// Mitsubishi GX Works2 project: 西松湘南道路1号機   PLC: Q03UDV
// 鹿島外環ロスゼロ

PROGRAM SIMLAT
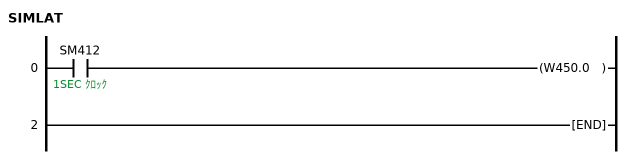
0     LD      SM412  ; 1SEC ｸﾛｯｸ
      OUT     W450.0
2     END
END_PROGRAM

PROGRAM FLEXPIWI
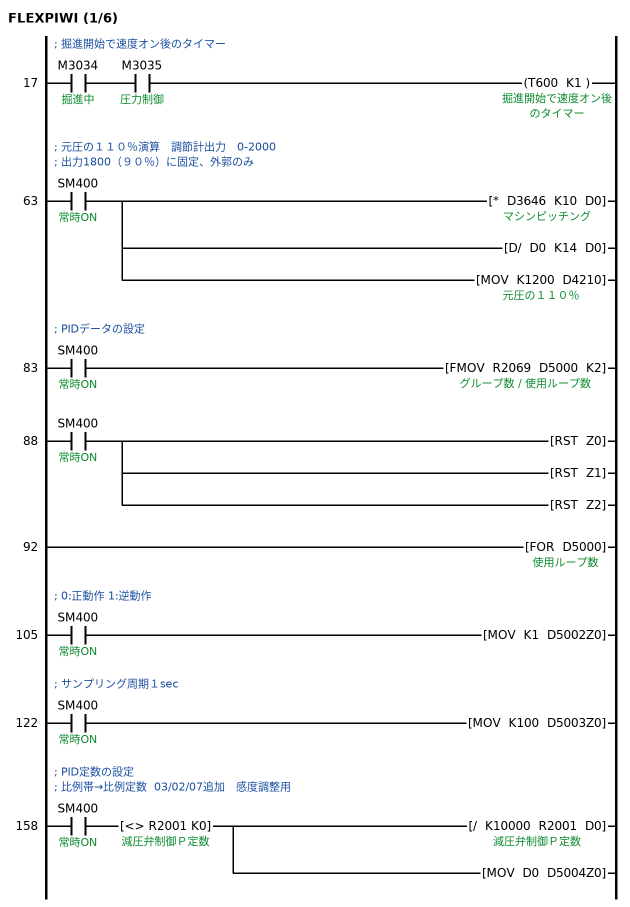
; 掘進開始で速度オン後のタイマー
17    LD      M3034  ; 掘進中
      AND     M3035  ; 圧力制御
      OUT     T600 K1  ; 掘進開始で速度オン後のタイマー
; 元圧の１１０％演算　調節計出力　0-2000
; 出力1800（９０％）に固定、外郭のみ
63    LD      SM400  ; 常時ON
      *       D3646 K10 D0  ; マシンピッチング
      D/      D0 K14 D0
      MOV     K1200 D4210  ; 元圧の１１０％
; PIDデータの設定
83    LD      SM400  ; 常時ON
      FMOV    R2069 D5000 K2  ; グループ数 / 使用ループ数
88    LD      SM400  ; 常時ON
      RST     Z0
      RST     Z1
      RST     Z2
92    FOR     D5000
; 0:正動作 1:逆動作
105   LD      SM400  ; 常時ON
      MOV     K1 D5002Z0
; サンプリング周期１sec
122   LD      SM400  ; 常時ON
      MOV     K100 D5003Z0
; PID定数の設定
; 比例帯→比例定数  03/02/07追加　感度調整用
158   LD      SM400  ; 常時ON
      AND<>   R2001 K0  ; 減圧弁制御Ｐ定数
      /       K10000 R2001 D0
      MOV     D0 D5004Z0
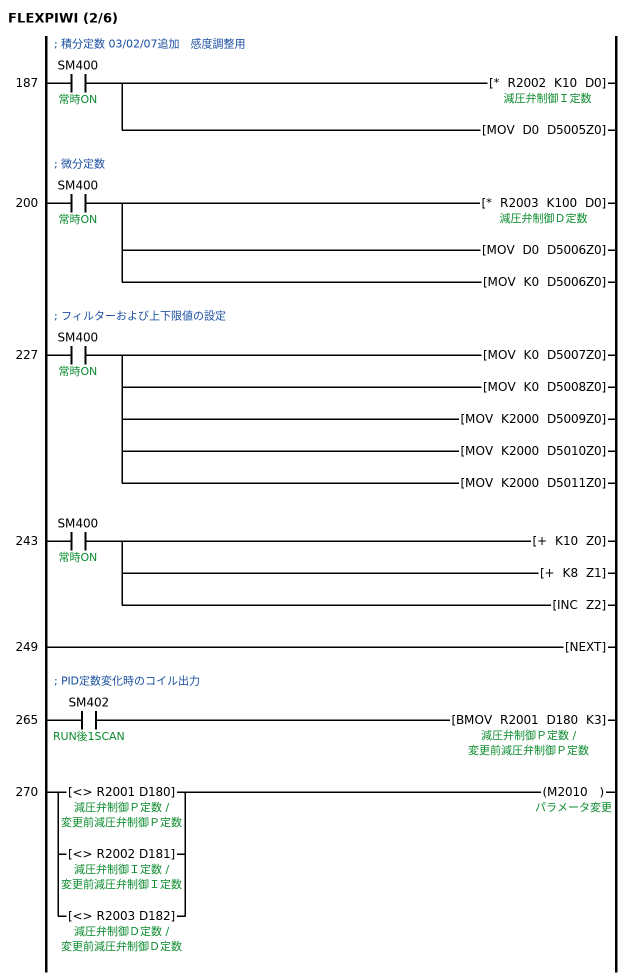
; 積分定数 03/02/07追加　感度調整用
187   LD      SM400  ; 常時ON
      *       R2002 K10 D0  ; 減圧弁制御Ｉ定数
      MOV     D0 D5005Z0
; 微分定数
200   LD      SM400  ; 常時ON
      *       R2003 K100 D0  ; 減圧弁制御Ｄ定数
      MOV     D0 D5006Z0
      MOV     K0 D5006Z0
; フィルターおよび上下限値の設定
227   LD      SM400  ; 常時ON
      MOV     K0 D5007Z0
      MOV     K0 D5008Z0
      MOV     K2000 D5009Z0
      MOV     K2000 D5010Z0
      MOV     K2000 D5011Z0
243   LD      SM400  ; 常時ON
      +       K10 Z0
      +       K8 Z1
      INC     Z2
249   NEXT
; PID定数変化時のコイル出力
265   LD      SM402  ; RUN後1SCAN
      BMOV    R2001 D180 K3  ; 変更前減圧弁制御Ｐ定数
270   LD<>    R2001 D180  ; 減圧弁制御Ｐ定数 / 変更前減圧弁制御Ｐ定数
      OR<>    R2002 D181  ; 減圧弁制御Ｉ定数 / 変更前減圧弁制御Ｉ定数
      OR<>    R2003 D182  ; 減圧弁制御Ｄ定数 / 変更前減圧弁制御Ｄ定数
      OUT     M2010  ; パラメータ変更
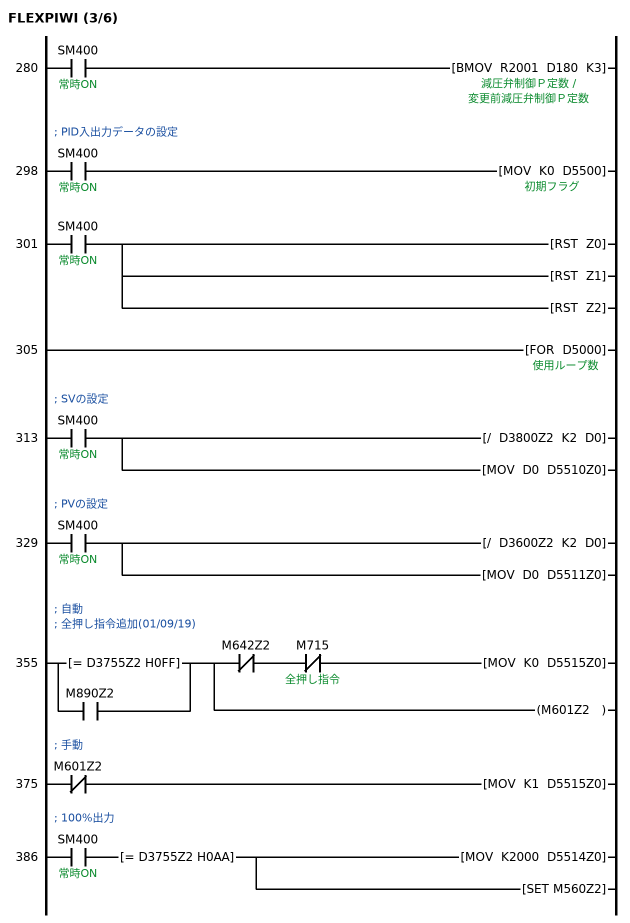
280   LD      SM400  ; 常時ON
      BMOV    R2001 D180 K3
; PID入出力データの設定
298   LD      SM400  ; 常時ON
      MOV     K0 D5500  ; 初期フラグ
301   LD      SM400  ; 常時ON
      RST     Z0
      RST     Z1
      RST     Z2
305   FOR     D5000
; SVの設定
313   LD      SM400  ; 常時ON
      /       D3800Z2 K2 D0
      MOV     D0 D5510Z0
; 
; PVの設定
329   LD      SM400  ; 常時ON
      /       D3600Z2 K2 D0
      MOV     D0 D5511Z0
; 自動
; 全押し指令追加(01/09/19)
355   LD=     D3755Z2 H0FF
      OR      M890Z2
      MPS
      ANI     M642Z2
      ANI     M715  ; 全押し指令
      MOV     K0 D5515Z0
      MPP
      OUT     M601Z2
; 手動
375   LDI     M601Z2
      MOV     K1 D5515Z0
; 100%出力
386   LD      SM400  ; 常時ON
      AND=    D3755Z2 H0AA
      MOV     K2000 D5514Z0
      SET     M560Z2
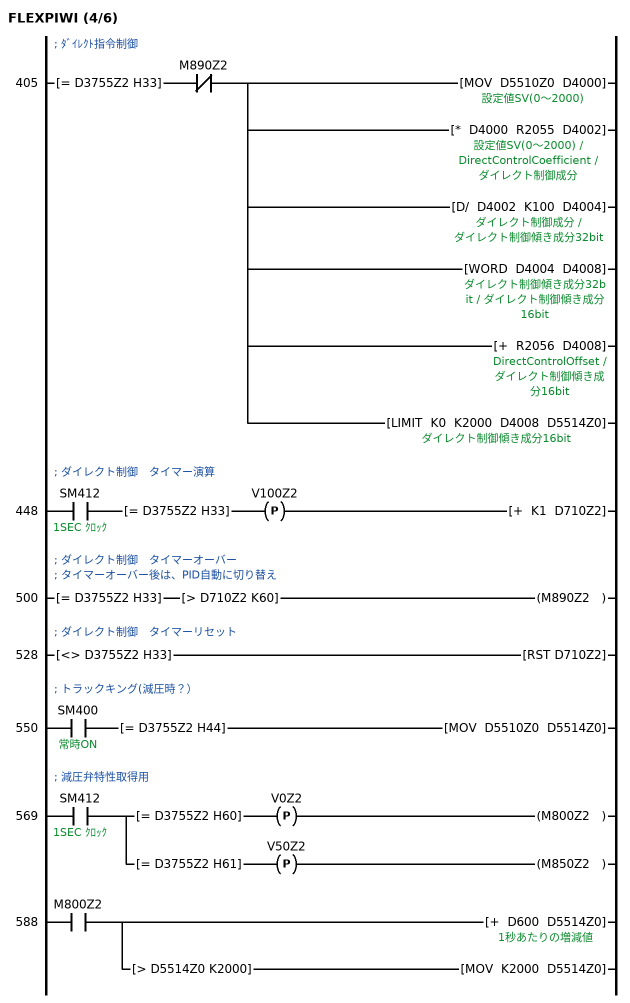
; ﾀﾞｲﾚｸﾄ指令制御
405   LD=     D3755Z2 H33
      ANI     M890Z2
      MOV     D5510Z0 D4000  ; 設定値SV(0～2000)
      *       D4000 R2055 D4002  ; DirectControlCoefficient / ダイレクト制御成分
      D/      D4002 K100 D4004  ; ダイレクト制御傾き成分32bit
      WORD    D4004 D4008  ; ダイレクト制御傾き成分16bit
      +       R2056 D4008  ; DirectControlOffset
      LIMIT   K0 K2000 D4008 D5514Z0
; ダイレクト制御　タイマー演算
448   LD      SM412  ; 1SEC ｸﾛｯｸ
      AND=    D3755Z2 H33
      EGP     V100Z2
      +       K1 D710Z2
; ダイレクト制御　タイマーオーバー
; タイマーオーバー後は、PID自動に切り替え
500   LD=     D3755Z2 H33
      AND>    D710Z2 K60
      OUT     M890Z2
; ダイレクト制御　タイマーリセット
528   LD<>    D3755Z2 H33
      RST     D710Z2
; トラックキング(減圧時？）
550   LD      SM400  ; 常時ON
      AND=    D3755Z2 H44
      MOV     D5510Z0 D5514Z0
; 減圧弁特性取得用
569   LD      SM412  ; 1SEC ｸﾛｯｸ
      MPS
      AND=    D3755Z2 H60
      EGP     V0Z2
      OUT     M800Z2
      MPP
      AND=    D3755Z2 H61
      EGP     V50Z2
      OUT     M850Z2
588   LD      M800Z2
      +       D600 D5514Z0  ; 1秒あたりの増減値
      AND>    D5514Z0 K2000
      MOV     K2000 D5514Z0
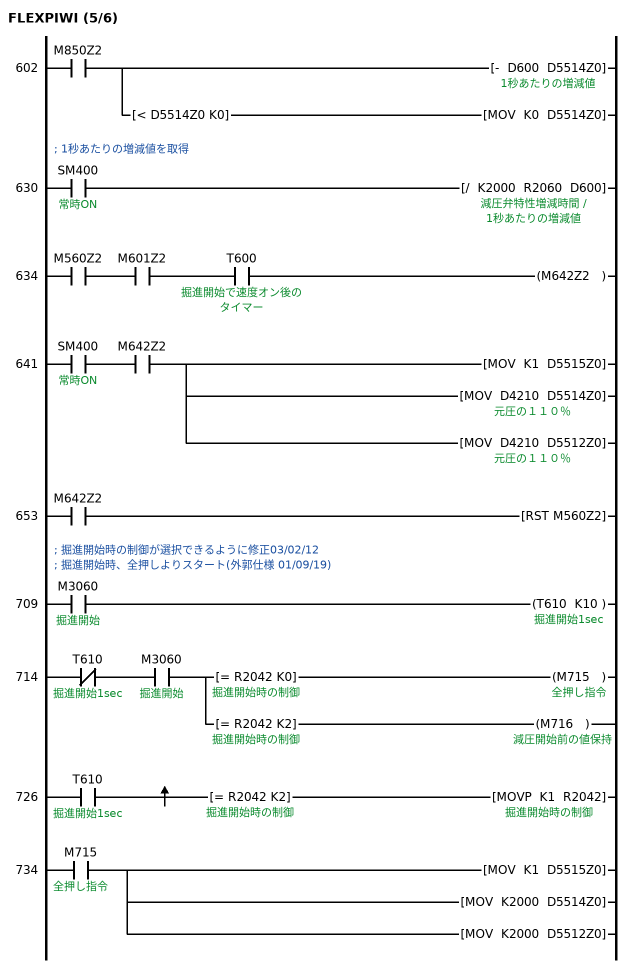
602   LD      M850Z2
      -       D600 D5514Z0
      AND<    D5514Z0 K0
      MOV     K0 D5514Z0
; 1秒あたりの増減値を取得
630   LD      SM400  ; 常時ON
      /       K2000 R2060 D600  ; 減圧弁特性増減時間
634   LD      M560Z2
      AND     M601Z2
      AND     T600  ; 掘進開始で速度オン後のタイマー
      OUT     M642Z2
641   LD      SM400  ; 常時ON
      AND     M642Z2
      MOV     K1 D5515Z0
      MOV     D4210 D5514Z0
      MOV     D4210 D5512Z0
653   LD      M642Z2
      RST     M560Z2
; 掘進開始時の制御が選択できるように修正03/02/12
; 掘進開始時、全押しよりスタート(外郭仕様 01/09/19)
709   LD      M3060  ; 掘進開始
      OUT     T610 K10  ; 掘進開始1sec
714   LDI     T610  ; 掘進開始1sec
      AND     M3060  ; 掘進開始
      MPS
      AND=    R2042 K0  ; 掘進開始時の制御
      OUT     M715  ; 全押し指令
      MPP
      AND=    R2042 K2  ; 掘進開始時の制御
      OUT     M716  ; 減圧開始前の値保持
726   LD      T610  ; 掘進開始1sec
      MEP
      AND=    R2042 K2  ; 掘進開始時の制御
      MOVP    K1 R2042
734   LD      M715  ; 全押し指令
      MOV     K1 D5515Z0
      MOV     K2000 D5514Z0
      MOV     K2000 D5512Z0
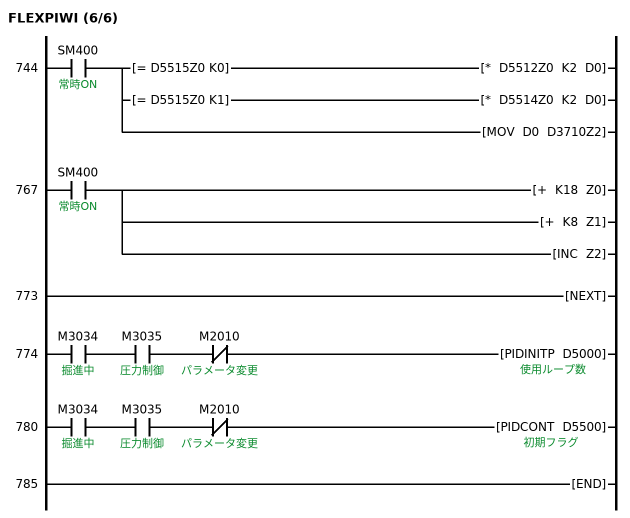
744   LD      SM400  ; 常時ON
      MPS
      AND=    D5515Z0 K0
      *       D5512Z0 K2 D0
      MRD
      AND=    D5515Z0 K1
      *       D5514Z0 K2 D0
      MPP
      MOV     D0 D3710Z2
767   LD      SM400  ; 常時ON
      +       K18 Z0
      +       K8 Z1
      INC     Z2
773   NEXT
774   LD      M3034  ; 掘進中
      AND     M3035  ; 圧力制御
      ANI     M2010  ; パラメータ変更
      PIDINITP D5000
780   LD      M3034  ; 掘進中
      AND     M3035  ; 圧力制御
      ANI     M2010  ; パラメータ変更
      PIDCONT D5500
785   END
END_PROGRAM

PROGRAM FLEXWIN
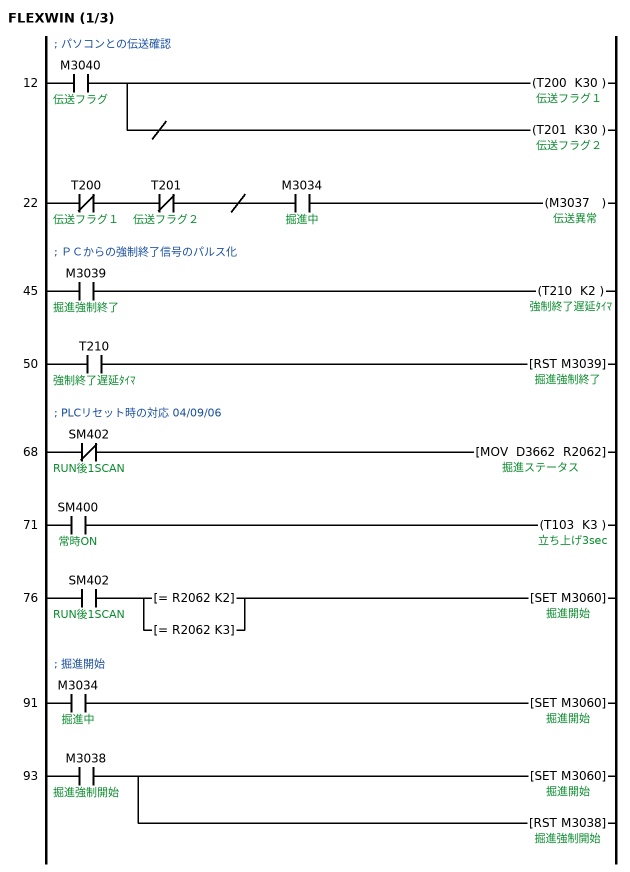
; パソコンとの伝送確認
12    LD      M3040  ; 伝送フラグ
      OUT     T200 K30  ; 伝送フラグ１
      INV
      OUT     T201 K30  ; 伝送フラグ２
22    LDI     T200  ; 伝送フラグ１
      ANI     T201  ; 伝送フラグ２
      INV
      AND     M3034  ; 掘進中
      OUT     M3037  ; 伝送異常
; ＰＣからの強制終了信号のパルス化
45    LD      M3039  ; 掘進強制終了
      OUT     T210 K2  ; 強制終了遅延ﾀｲﾏ
50    LD      T210  ; 強制終了遅延ﾀｲﾏ
      RST     M3039  ; 掘進強制終了
; PLCリセット時の対応 04/09/06
68    LDI     SM402  ; RUN後1SCAN
      MOV     D3662 R2062  ; 掘進ステータス
71    LD      SM400  ; 常時ON
      OUT     T103 K3  ; 立ち上げ3sec
76    LD      SM402  ; RUN後1SCAN
      LD=     R2062 K2
      OR=     R2062 K3
      ANB
      SET     M3060  ; 掘進開始
; 掘進開始
91    LD      M3034  ; 掘進中
      SET     M3060  ; 掘進開始
93    LD      M3038  ; 掘進強制開始
      SET     M3060  ; 掘進開始
      RST     M3038  ; 掘進強制開始
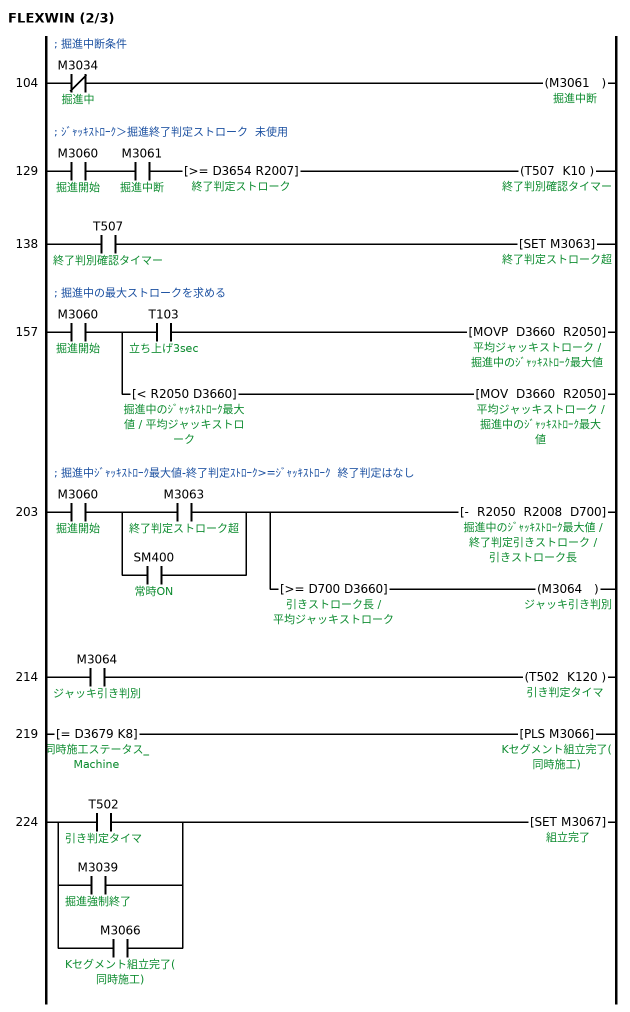
; 掘進中断条件
104   LDI     M3034  ; 掘進中
      OUT     M3061  ; 掘進中断
; ｼﾞｬｯｷｽﾄﾛｰｸ＞掘進終了判定ストローク  未使用
129   LD      M3060  ; 掘進開始
      AND     M3061  ; 掘進中断
      AND>=   D3654 R2007  ; 終了判定ストローク
      OUT     T507 K10  ; 終了判別確認タイマー
138   LD      T507  ; 終了判別確認タイマー
      SET     M3063  ; 終了判定ストローク超
; 掘進中の最大ストロークを求める
157   LD      M3060  ; 掘進開始
      MPS
      AND     T103  ; 立ち上げ3sec
      MOVP    D3660 R2050  ; 平均ジャッキストローク / 掘進中のｼﾞｬｯｷｽﾄﾛｰｸ最大値
      MPP
      AND<    R2050 D3660  ; 掘進中のｼﾞｬｯｷｽﾄﾛｰｸ最大値 / 平均ジャッキストローク
      MOV     D3660 R2050
; 掘進中ｼﾞｬｯｷｽﾄﾛｰｸ最大値-終了判定ｽﾄﾛｰｸ>=ｼﾞｬｯｷｽﾄﾛｰｸ  終了判定はなし
203   LD      M3060  ; 掘進開始
      LD      M3063  ; 終了判定ストローク超
      OR      SM400  ; 常時ON
      ANB
      -       R2050 R2008 D700  ; 終了判定引きストローク / 引きストローク長
      AND>=   D700 D3660  ; 引きストローク長 / 平均ジャッキストローク
      OUT     M3064  ; ジャッキ引き判別
214   LD      M3064  ; ジャッキ引き判別
      OUT     T502 K120  ; 引き判定タイマ
219   LD=     D3679 K8  ; 同時施工ステータス_Machine
      PLS     M3066  ; Kセグメント組立完了(同時施工)
224   LD      T502  ; 引き判定タイマ
      OR      M3039  ; 掘進強制終了
      OR      M3066  ; Kセグメント組立完了(同時施工)
      SET     M3067  ; 組立完了
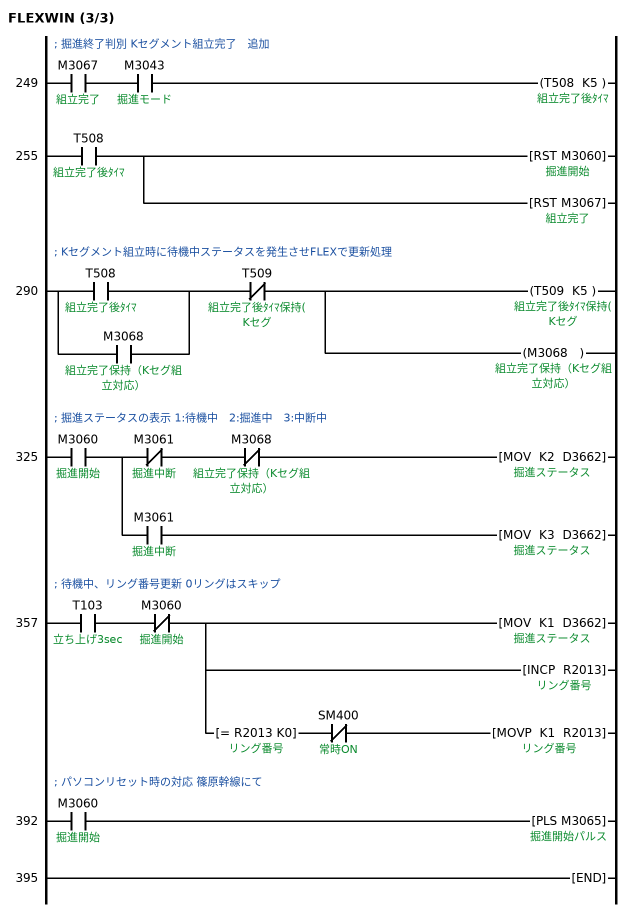
; 掘進終了判別 Kセグメント組立完了　追加
249   LD      M3067  ; 組立完了
      AND     M3043  ; 掘進モード
      OUT     T508 K5  ; 組立完了後ﾀｲﾏ
255   LD      T508  ; 組立完了後ﾀｲﾏ
      RST     M3060  ; 掘進開始
      RST     M3067  ; 組立完了
; Kセグメント組立時に待機中ステータスを発生させFLEXで更新処理
290   LD      T508  ; 組立完了後ﾀｲﾏ
      OR      M3068  ; 組立完了保持（Kセグ組立対応）
      ANI     T509  ; 組立完了後ﾀｲﾏ保持(Kセグ
      OUT     T509 K5  ; 組立完了後ﾀｲﾏ保持(Kセグ
      OUT     M3068  ; 組立完了保持（Kセグ組立対応）
; 掘進ステータスの表示 1:待機中　2:掘進中　3:中断中
325   LD      M3060  ; 掘進開始
      MPS
      ANI     M3061  ; 掘進中断
      ANI     M3068  ; 組立完了保持（Kセグ組立対応）
      MOV     K2 D3662
      MPP
      AND     M3061  ; 掘進中断
      MOV     K3 D3662
; 待機中、リング番号更新 0リングはスキップ
357   LD      T103  ; 立ち上げ3sec
      ANI     M3060  ; 掘進開始
      MOV     K1 D3662
      INCP    R2013  ; リング番号
      AND=    R2013 K0  ; リング番号
      ANI     SM400  ; 常時ON
      MOVP    K1 R2013
; パソコンリセット時の対応 篠原幹線にて
392   LD      M3060  ; 掘進開始
      PLS     M3065  ; 掘進開始パルス
395   END
END_PROGRAM

PROGRAM INOUTWIN  // 西松湘南道路1号機
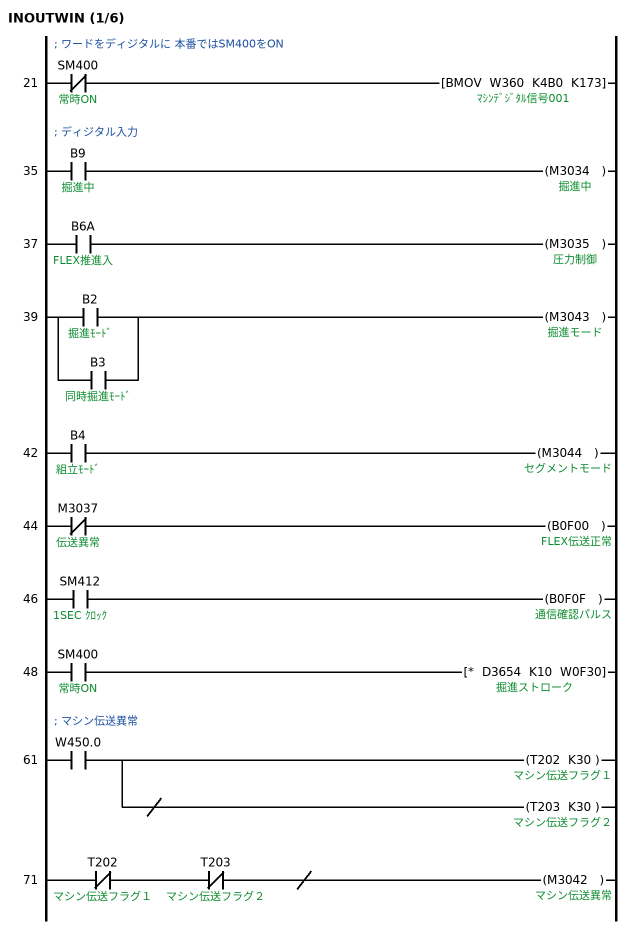
; ワードをディジタルに 本番ではSM400をON
21    LDI     SM400  ; 常時ON
      BMOV    W360 K4B0 K173  ; ﾏｼﾝﾃﾞｼﾞﾀﾙ信号001 / 中央操作
; ディジタル入力
35    LD      B9  ; 掘進中
      OUT     M3034  ; 掘進中
37    LD      B6A  ; FLEX推進入
      OUT     M3035  ; 圧力制御
39    LD      B2  ; 掘進ﾓｰﾄﾞ
      OR      B3  ; 同時掘進ﾓｰﾄﾞ
      OUT     M3043  ; 掘進モード
42    LD      B4  ; 組立ﾓｰﾄﾞ
      OUT     M3044  ; セグメントモード
44    LDI     M3037  ; 伝送異常
      OUT     B0F00  ; FLEX伝送正常
46    LD      SM412  ; 1SEC ｸﾛｯｸ
      OUT     B0F0F  ; 通信確認パルス
48    LD      SM400  ; 常時ON
      *       D3654 K10 W0F30  ; 掘進ストローク
; マシン伝送異常
61    LD      W450.0
      OUT     T202 K30  ; マシン伝送フラグ１
      INV
      OUT     T203 K30  ; マシン伝送フラグ２
71    LDI     T202  ; マシン伝送フラグ１
      ANI     T203  ; マシン伝送フラグ２
      INV
      OUT     M3042  ; マシン伝送異常
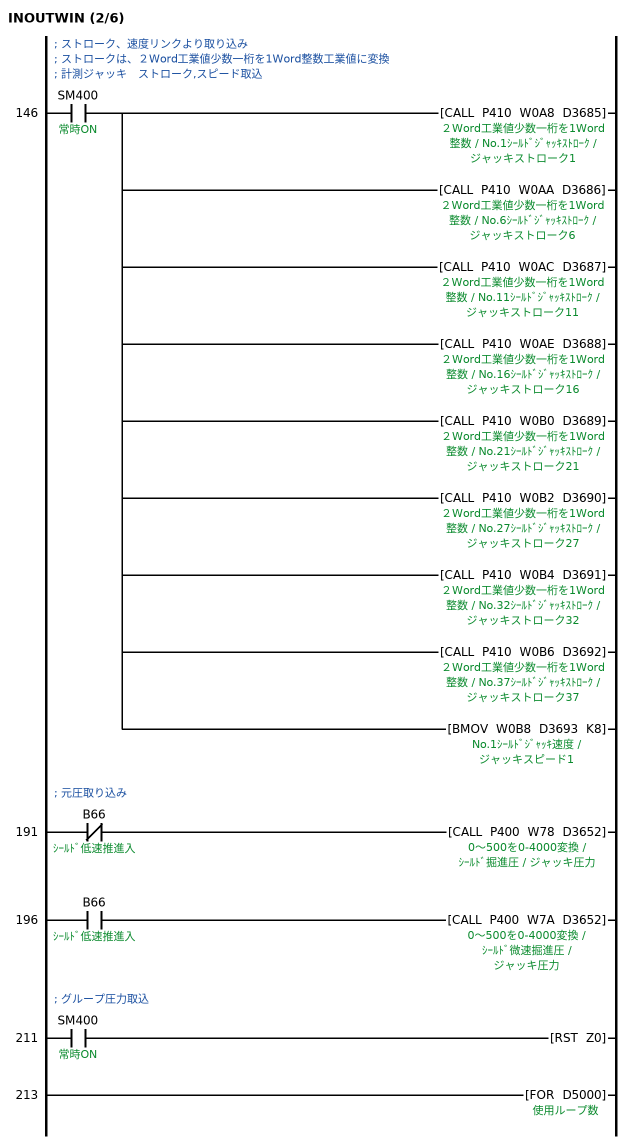
; ストローク、速度リンクより取り込み
; ストロークは、２Word工業値少数一桁を1Word整数工業値に変換
; 計測ジャッキ　ストローク,スピード取込
146   LD      SM400  ; 常時ON
      CALL    P410 W0A8 D3685  ; ２Word工業値少数一桁を1Word整数 / No.1ｼｰﾙﾄﾞｼﾞｬｯｷｽﾄﾛｰｸ / ジャッキストローク1
      CALL    P410 W0AA D3686  ; No.6ｼｰﾙﾄﾞｼﾞｬｯｷｽﾄﾛｰｸ / ジャッキストローク6
      CALL    P410 W0AC D3687  ; No.11ｼｰﾙﾄﾞｼﾞｬｯｷｽﾄﾛｰｸ / ジャッキストローク11
      CALL    P410 W0AE D3688  ; No.16ｼｰﾙﾄﾞｼﾞｬｯｷｽﾄﾛｰｸ / ジャッキストローク16
      CALL    P410 W0B0 D3689  ; No.21ｼｰﾙﾄﾞｼﾞｬｯｷｽﾄﾛｰｸ / ジャッキストローク21
      CALL    P410 W0B2 D3690  ; No.27ｼｰﾙﾄﾞｼﾞｬｯｷｽﾄﾛｰｸ / ジャッキストローク27
      CALL    P410 W0B4 D3691  ; No.32ｼｰﾙﾄﾞｼﾞｬｯｷｽﾄﾛｰｸ / ジャッキストローク32
      CALL    P410 W0B6 D3692  ; No.37ｼｰﾙﾄﾞｼﾞｬｯｷｽﾄﾛｰｸ / ジャッキストローク37
      BMOV    W0B8 D3693 K8  ; No.1ｼｰﾙﾄﾞｼﾞｬｯｷ速度 / ジャッキスピード1
; 元圧取り込み
191   LDI     B66  ; ｼｰﾙﾄﾞ低速推進入
      CALL    P400 W78 D3652  ; 0～500を0-4000変換 / ｼｰﾙﾄﾞ掘進圧 / ジャッキ圧力
196   LD      B66  ; ｼｰﾙﾄﾞ低速推進入
      CALL    P400 W7A D3652  ; ｼｰﾙﾄﾞ微速掘進圧
; グループ圧力取込
211   LD      SM400  ; 常時ON
      RST     Z0
213   FOR     D5000  ; 使用ループ数
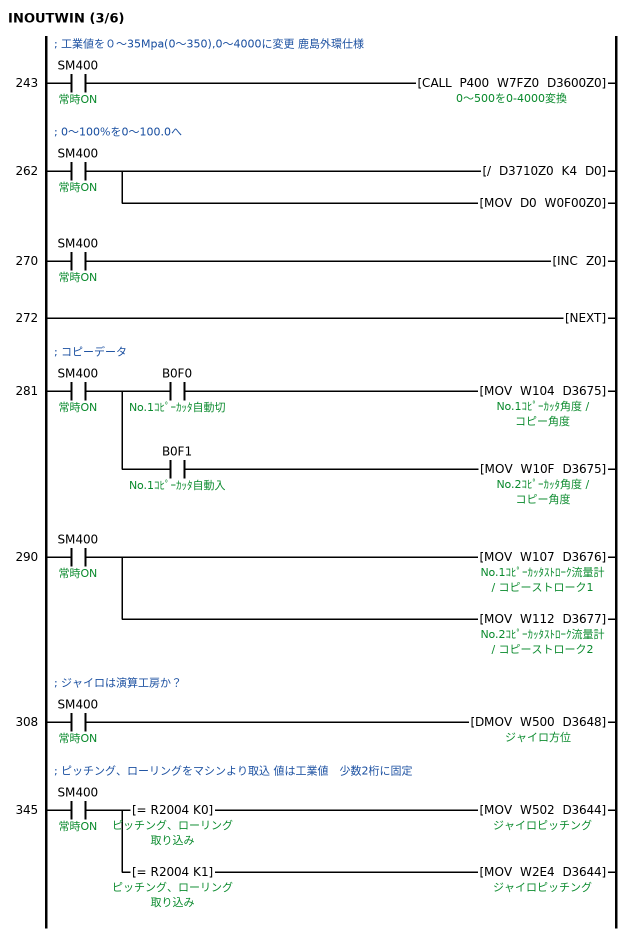
; 工業値を０～35Mpa(0～350),0～4000に変更 鹿島外環仕様
243   LD      SM400  ; 常時ON
      CALL    P400 W7FZ0 D3600Z0
; 0～100%を0～100.0へ
262   LD      SM400  ; 常時ON
      /       D3710Z0 K4 D0
      MOV     D0 W0F00Z0
270   LD      SM400  ; 常時ON
      INC     Z0
272   NEXT
; コピーデータ
281   LD      SM400  ; 常時ON
      MPS
      AND     B0F0  ; No.1ｺﾋﾟｰｶｯﾀ自動切
      MOV     W104 D3675  ; No.1ｺﾋﾟｰｶｯﾀ角度 / コピー角度
      MPP
      AND     B0F1  ; No.1ｺﾋﾟｰｶｯﾀ自動入
      MOV     W10F D3675  ; No.2ｺﾋﾟｰｶｯﾀ角度
290   LD      SM400  ; 常時ON
      MOV     W107 D3676  ; No.1ｺﾋﾟｰｶｯﾀｽﾄﾛｰｸ流量計 / コピーストローク1
      MOV     W112 D3677  ; No.2ｺﾋﾟｰｶｯﾀｽﾄﾛｰｸ流量計 / コピーストローク2
; ジャイロは演算工房か？
308   LD      SM400  ; 常時ON
      DMOV    W500 D3648  ; ジャイロ方位
; ピッチング、ローリングをマシンより取込 値は工業値　少数2桁に固定
345   LD      SM400  ; 常時ON
      MPS
      AND=    R2004 K0  ; ピッチング、ローリング取り込み
      MOV     W502 D3644  ; ジャイロピッチング
      MPP
      AND=    R2004 K1  ; ピッチング、ローリング取り込み
      MOV     W2E4 D3644
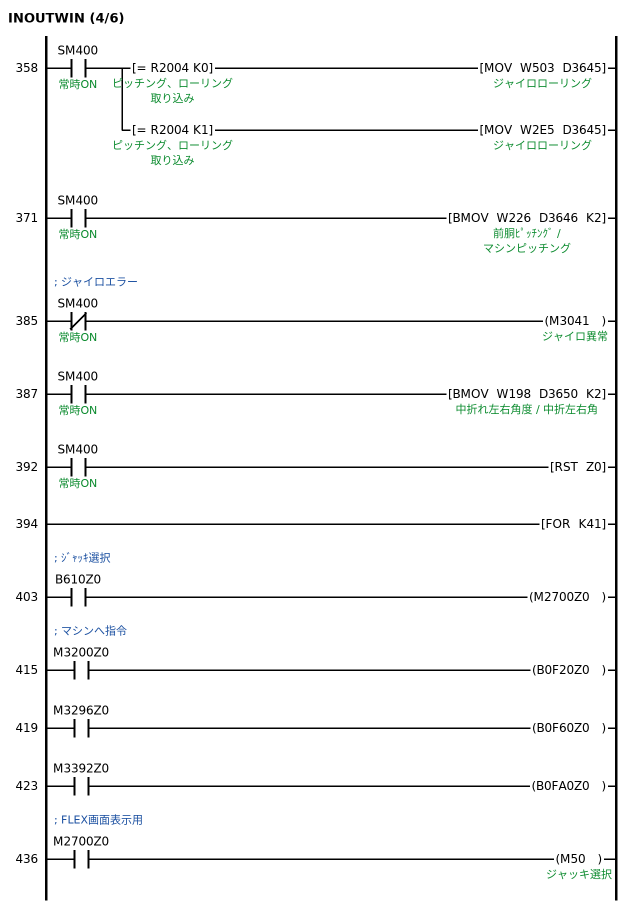
358   LD      SM400  ; 常時ON
      MPS
      AND=    R2004 K0  ; ピッチング、ローリング取り込み
      MOV     W503 D3645  ; ジャイロローリング
      MPP
      AND=    R2004 K1  ; ピッチング、ローリング取り込み
      MOV     W2E5 D3645
371   LD      SM400  ; 常時ON
      BMOV    W226 D3646 K2  ; 前胴ﾋﾟｯﾁﾝｸﾞ / マシンピッチング
; ジャイロエラー
385   LDI     SM400  ; 常時ON
      OUT     M3041  ; ジャイロ異常
387   LD      SM400  ; 常時ON
      BMOV    W198 D3650 K2  ; 中折れ左右角度 / 中折左右角
392   LD      SM400  ; 常時ON
      RST     Z0
394   FOR     K41
; ｼﾞｬｯｷ選択
403   LD      B610Z0
      OUT     M2700Z0
; マシンへ指令
415   LD      M3200Z0
      OUT     B0F20Z0
419   LD      M3296Z0
      OUT     B0F60Z0
423   LD      M3392Z0
      OUT     B0FA0Z0
; FLEX画面表示用
436   LD      M2700Z0
      OUT     M50  ; ジャッキ選択
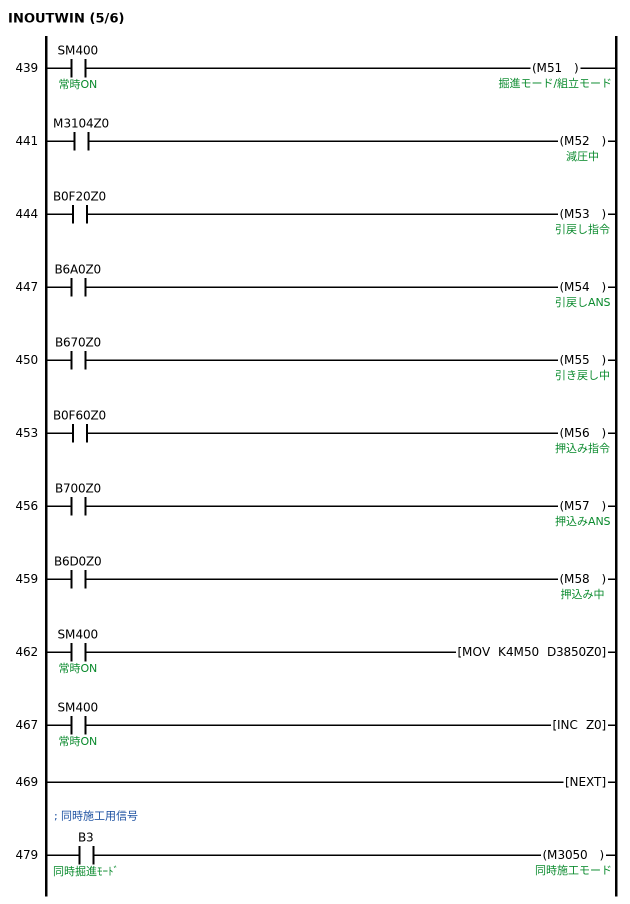
439   LD      SM400  ; 常時ON
      OUT     M51  ; 掘進モード/組立モード
441   LD      M3104Z0
      OUT     M52  ; 減圧中
444   LD      B0F20Z0
      OUT     M53  ; 引戻し指令
447   LD      B6A0Z0
      OUT     M54  ; 引戻しANS
450   LD      B670Z0
      OUT     M55  ; 引き戻し中
453   LD      B0F60Z0
      OUT     M56  ; 押込み指令
456   LD      B700Z0
      OUT     M57  ; 押込みANS
459   LD      B6D0Z0
      OUT     M58  ; 押込み中
462   LD      SM400  ; 常時ON
      MOV     K4M50 D3850Z0
467   LD      SM400  ; 常時ON
      INC     Z0
469   NEXT
; 同時施工用信号
479   LD      B3  ; 同時掘進ﾓｰﾄﾞ
      OUT     M3050  ; 同時施工モード
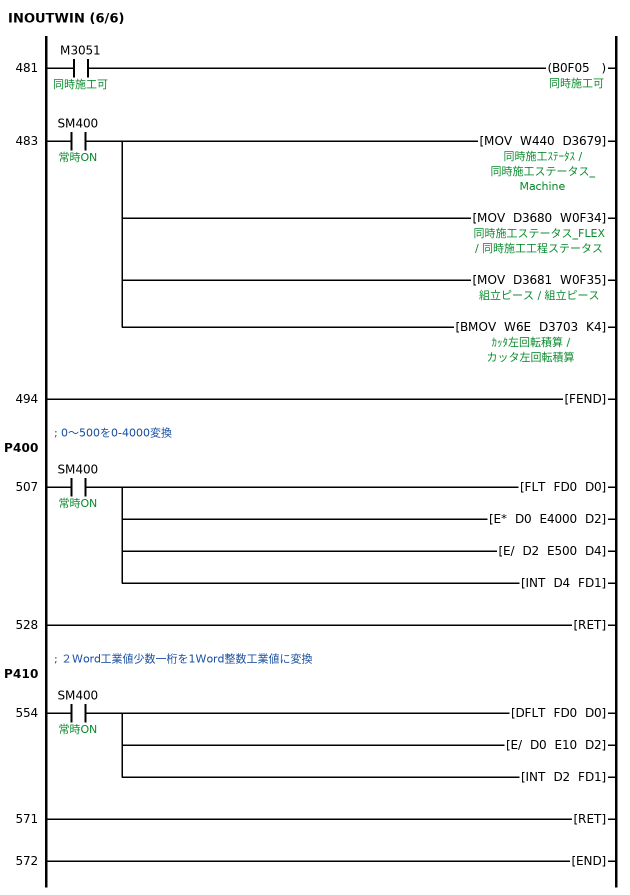
481   LD      M3051  ; 同時施工可
      OUT     B0F05  ; 同時施工可
483   LD      SM400  ; 常時ON
      MOV     W440 D3679  ; 同時施工ｽﾃｰﾀｽ / 同時施工ステータス_Machine
      MOV     D3680 W0F34  ; 同時施工ステータス_FLEX / 同時施工工程ステータス
      MOV     D3681 W0F35  ; 組立ピース / 組立ピース
      BMOV    W6E D3703 K4  ; ｶｯﾀ左回転積算 / カッタ左回転積算
494   FEND
      P400
; 0～500を0-4000変換
507   LD      SM400  ; 常時ON
      FLT     FD0 D0
        [note] スケール上限
      E*      D0 E4000 D2
      E/      D2 E500 D4
      INT     D4 FD1
528   RET
      P410
; ２Word工業値少数一桁を1Word整数工業値に変換
554   LD      SM400  ; 常時ON
      DFLT    FD0 D0
        [note] スケール上限
      E/      D0 E10 D2
      INT     D2 FD1
571   RET
572   END
END_PROGRAM

// device comments not shown above
D710  ; グループ1ダイレクト時間
D3600  ; グループ1圧力
D3710  ; グループ1圧力MV
D3800  ; グループ1圧力SV
D5512  ; グループ1自動操作量（MV)
D5514  ; グループ1手動操作量（MV)
